{attribute addProperty BoxType "EL3058-0000-0017"}
{attribute addProperty Id "AI_Standard_ChannelAT %I*ARRAY[0..7] OF AI_Standard_Channel_B51B79FC648810WcStateAT %I*WcState_F855686C1620InfoDataAT %I*InfoData_BC63D37F80100"}
{attribute addProperty CRC "1638664833"}
{attribute addProperty SizeInBites "744"}
{attribute addProperty SizeInBytes "93"}
TYPE EL3058_D68B7A11 :
STRUCT
	{attribute addProperty Name "AI_Standard_Channel"}
	AI_Standard_Channel : ARRAY[0..7] OF AI_Standard_Channel_B51B79FC;
	{attribute addProperty Name "WcState"}
	WcState : WcState_F855686C;
	{attribute addProperty Name "InfoData"}
	InfoData : InfoData_BC63D37F;
END_STRUCT
END_TYPE

(* stored: Version 1.2.0.0, ProductVersion 3.1.4024.9
   DUT EL3058_D68B7A11: Id {6ed01f1c-2d44-481f-a62f-acc7115c6ac2} *)
